{attribute addProperty BoxType "KL2631"}
{attribute addProperty Id "Channel_1Channel_E75BD82E00"}
{attribute addProperty CRC "475127576"}
{attribute addProperty SizeInBites "0"}
{attribute addProperty SizeInBytes "0"}
TYPE KL2631_1C51DF18 :
STRUCT
	{attribute addProperty Name "Channel_1"}
	Channel_1 : Channel_E75BD82E;
END_STRUCT
END_TYPE

(* stored: Version 1.2.0.0, ProductVersion 3.1.4024.9
   DUT KL2631_1C51DF18: Id {8b5e6f20-f52a-4183-85fa-01f91feb953b} *)
